{attribute 'pack_mode' := '1'}
TYPE Fan :
STRUCT
	nSpeed 	: INT; // control primary fan speed 0-100%
	nTemp	: INT; // prim fan's terminal temp in Celcius
	fFE		: REAL;
END_STRUCT
END_TYPE

(* stored: Version 1.1.0.1, ProductVersion 3.1.4022.18
   DUT Fan: Id {9a2dd2f8-0729-4a1c-bace-ed9eff5a0ecb} *)
